{attribute 'qualified_only'}
{attribute 'TcContextName':='SerialComTask'} //the variables in this lib are sync with the SerialComTask
VAR_GLOBAL
	fbStim300 : ARRAY [0..2] OF FB_MapStim300;	
END_VAR

(* stored: Version 1.1.0.1, ProductVersion 3.1.4024.9
   GVL IMU: Id {c8ca64f0-43cf-46d6-826e-3cf6b4689ec3} *)
